FUNCTION_BLOCK Unifilar_HMI (* Service Interface Function Block Type *)
  (* Standard: 61499-2 *)
  (* Version 0.0, 21/04/2026, template *)
  PACKAGE Hidryco.HidrycoLib;
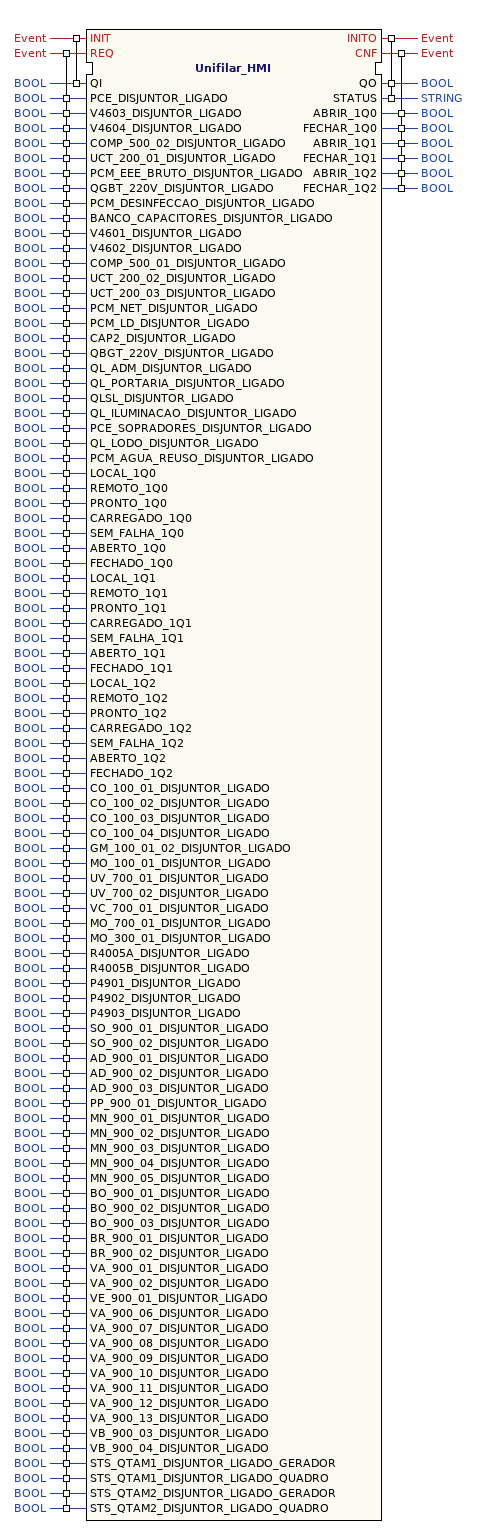
  EVENT_INPUT
    INIT WITH QI;
    REQ WITH PCE_DISJUNTOR_LIGADO, V4603_DISJUNTOR_LIGADO, V4604_DISJUNTOR_LIGADO, COMP_500_02_DISJUNTOR_LIGADO, UCT_200_01_DISJUNTOR_LIGADO, PCM_EEE_BRUTO_DISJUNTOR_LIGADO, QGBT_220V_DISJUNTOR_LIGADO, PCM_DESINFECCAO_DISJUNTOR_LIGADO, BANCO_CAPACITORES_DISJUNTOR_LIGADO, V4601_DISJUNTOR_LIGADO, V4602_DISJUNTOR_LIGADO, COMP_500_01_DISJUNTOR_LIGADO, UCT_200_02_DISJUNTOR_LIGADO, UCT_200_03_DISJUNTOR_LIGADO, PCM_NET_DISJUNTOR_LIGADO, PCM_LD_DISJUNTOR_LIGADO, CAP2_DISJUNTOR_LIGADO, QBGT_220V_DISJUNTOR_LIGADO, QL_ADM_DISJUNTOR_LIGADO, QL_PORTARIA_DISJUNTOR_LIGADO, QLSL_DISJUNTOR_LIGADO, QL_ILUMINACAO_DISJUNTOR_LIGADO, PCE_SOPRADORES_DISJUNTOR_LIGADO, QL_LODO_DISJUNTOR_LIGADO, PCM_AGUA_REUSO_DISJUNTOR_LIGADO, LOCAL_1Q0, REMOTO_1Q0, PRONTO_1Q0, CARREGADO_1Q0, SEM_FALHA_1Q0, ABERTO_1Q0, FECHADO_1Q0, LOCAL_1Q1, REMOTO_1Q1, PRONTO_1Q1, CARREGADO_1Q1, SEM_FALHA_1Q1, ABERTO_1Q1, FECHADO_1Q1, LOCAL_1Q2, REMOTO_1Q2, PRONTO_1Q2, CARREGADO_1Q2, SEM_FALHA_1Q2, ABERTO_1Q2, FECHADO_1Q2, CO_100_01_DISJUNTOR_LIGADO, CO_100_02_DISJUNTOR_LIGADO, CO_100_03_DISJUNTOR_LIGADO, CO_100_04_DISJUNTOR_LIGADO, GM_100_01_02_DISJUNTOR_LIGADO, MO_100_01_DISJUNTOR_LIGADO, UV_700_01_DISJUNTOR_LIGADO, UV_700_02_DISJUNTOR_LIGADO, VC_700_01_DISJUNTOR_LIGADO, MO_700_01_DISJUNTOR_LIGADO, MO_300_01_DISJUNTOR_LIGADO, R4005A_DISJUNTOR_LIGADO, R4005B_DISJUNTOR_LIGADO, P4901_DISJUNTOR_LIGADO, P4902_DISJUNTOR_LIGADO, P4903_DISJUNTOR_LIGADO, SO_900_01_DISJUNTOR_LIGADO, SO_900_02_DISJUNTOR_LIGADO, AD_900_01_DISJUNTOR_LIGADO, AD_900_02_DISJUNTOR_LIGADO, AD_900_03_DISJUNTOR_LIGADO, PP_900_01_DISJUNTOR_LIGADO, MN_900_01_DISJUNTOR_LIGADO, MN_900_02_DISJUNTOR_LIGADO, MN_900_03_DISJUNTOR_LIGADO, MN_900_04_DISJUNTOR_LIGADO, MN_900_05_DISJUNTOR_LIGADO, BO_900_01_DISJUNTOR_LIGADO, BO_900_02_DISJUNTOR_LIGADO, BO_900_03_DISJUNTOR_LIGADO, BR_900_01_DISJUNTOR_LIGADO, BR_900_02_DISJUNTOR_LIGADO, VA_900_01_DISJUNTOR_LIGADO, VA_900_02_DISJUNTOR_LIGADO, VE_900_01_DISJUNTOR_LIGADO, VA_900_06_DISJUNTOR_LIGADO, VA_900_07_DISJUNTOR_LIGADO, VA_900_08_DISJUNTOR_LIGADO, VA_900_09_DISJUNTOR_LIGADO, VA_900_10_DISJUNTOR_LIGADO, VA_900_11_DISJUNTOR_LIGADO, VA_900_12_DISJUNTOR_LIGADO, VA_900_13_DISJUNTOR_LIGADO, VB_900_03_DISJUNTOR_LIGADO, VB_900_04_DISJUNTOR_LIGADO, STS_QTAM1_DISJUNTOR_LIGADO_GERADOR, STS_QTAM1_DISJUNTOR_LIGADO_QUADRO, STS_QTAM2_DISJUNTOR_LIGADO_GERADOR, STS_QTAM2_DISJUNTOR_LIGADO_QUADRO;
  END_EVENT
  EVENT_OUTPUT
    INITO WITH QO, STATUS;
    CNF WITH ABRIR_1Q0, FECHAR_1Q0, ABRIR_1Q1, FECHAR_1Q1, ABRIR_1Q2, FECHAR_1Q2;
  END_EVENT
  VAR_INPUT
    QI : BOOL;
    PCE_DISJUNTOR_LIGADO : BOOL;
    V4603_DISJUNTOR_LIGADO : BOOL;
    V4604_DISJUNTOR_LIGADO : BOOL;
    COMP_500_02_DISJUNTOR_LIGADO : BOOL;
    UCT_200_01_DISJUNTOR_LIGADO : BOOL;
    PCM_EEE_BRUTO_DISJUNTOR_LIGADO : BOOL;
    QGBT_220V_DISJUNTOR_LIGADO : BOOL;
    PCM_DESINFECCAO_DISJUNTOR_LIGADO : BOOL;
    BANCO_CAPACITORES_DISJUNTOR_LIGADO : BOOL;
    V4601_DISJUNTOR_LIGADO : BOOL;
    V4602_DISJUNTOR_LIGADO : BOOL;
    COMP_500_01_DISJUNTOR_LIGADO : BOOL;
    UCT_200_02_DISJUNTOR_LIGADO : BOOL;
    UCT_200_03_DISJUNTOR_LIGADO : BOOL;
    PCM_NET_DISJUNTOR_LIGADO : BOOL;
    PCM_LD_DISJUNTOR_LIGADO : BOOL;
    CAP2_DISJUNTOR_LIGADO : BOOL;
    QBGT_220V_DISJUNTOR_LIGADO : BOOL;
    QL_ADM_DISJUNTOR_LIGADO : BOOL;
    QL_PORTARIA_DISJUNTOR_LIGADO : BOOL;
    QLSL_DISJUNTOR_LIGADO : BOOL;
    QL_ILUMINACAO_DISJUNTOR_LIGADO : BOOL;
    PCE_SOPRADORES_DISJUNTOR_LIGADO : BOOL;
    QL_LODO_DISJUNTOR_LIGADO : BOOL;
    PCM_AGUA_REUSO_DISJUNTOR_LIGADO : BOOL;
    LOCAL_1Q0 : BOOL;
    REMOTO_1Q0 : BOOL;
    PRONTO_1Q0 : BOOL;
    CARREGADO_1Q0 : BOOL;
    SEM_FALHA_1Q0 : BOOL;
    ABERTO_1Q0 : BOOL;
    FECHADO_1Q0 : BOOL;
    LOCAL_1Q1 : BOOL;
    REMOTO_1Q1 : BOOL;
    PRONTO_1Q1 : BOOL;
    CARREGADO_1Q1 : BOOL;
    SEM_FALHA_1Q1 : BOOL;
    ABERTO_1Q1 : BOOL;
    FECHADO_1Q1 : BOOL;
    LOCAL_1Q2 : BOOL;
    REMOTO_1Q2 : BOOL;
    PRONTO_1Q2 : BOOL;
    CARREGADO_1Q2 : BOOL;
    SEM_FALHA_1Q2 : BOOL;
    ABERTO_1Q2 : BOOL;
    FECHADO_1Q2 : BOOL;
    CO_100_01_DISJUNTOR_LIGADO : BOOL;
    CO_100_02_DISJUNTOR_LIGADO : BOOL;
    CO_100_03_DISJUNTOR_LIGADO : BOOL;
    CO_100_04_DISJUNTOR_LIGADO : BOOL;
    GM_100_01_02_DISJUNTOR_LIGADO : BOOL;
    MO_100_01_DISJUNTOR_LIGADO : BOOL;
    UV_700_01_DISJUNTOR_LIGADO : BOOL;
    UV_700_02_DISJUNTOR_LIGADO : BOOL;
    VC_700_01_DISJUNTOR_LIGADO : BOOL;
    MO_700_01_DISJUNTOR_LIGADO : BOOL;
    MO_300_01_DISJUNTOR_LIGADO : BOOL;
    R4005A_DISJUNTOR_LIGADO : BOOL;
    R4005B_DISJUNTOR_LIGADO : BOOL;
    P4901_DISJUNTOR_LIGADO : BOOL;
    P4902_DISJUNTOR_LIGADO : BOOL;
    P4903_DISJUNTOR_LIGADO : BOOL;
    SO_900_01_DISJUNTOR_LIGADO : BOOL;
    SO_900_02_DISJUNTOR_LIGADO : BOOL;
    AD_900_01_DISJUNTOR_LIGADO : BOOL;
    AD_900_02_DISJUNTOR_LIGADO : BOOL;
    AD_900_03_DISJUNTOR_LIGADO : BOOL;
    PP_900_01_DISJUNTOR_LIGADO : BOOL;
    MN_900_01_DISJUNTOR_LIGADO : BOOL;
    MN_900_02_DISJUNTOR_LIGADO : BOOL;
    MN_900_03_DISJUNTOR_LIGADO : BOOL;
    MN_900_04_DISJUNTOR_LIGADO : BOOL;
    MN_900_05_DISJUNTOR_LIGADO : BOOL;
    BO_900_01_DISJUNTOR_LIGADO : BOOL;
    BO_900_02_DISJUNTOR_LIGADO : BOOL;
    BO_900_03_DISJUNTOR_LIGADO : BOOL;
    BR_900_01_DISJUNTOR_LIGADO : BOOL;
    BR_900_02_DISJUNTOR_LIGADO : BOOL;
    VA_900_01_DISJUNTOR_LIGADO : BOOL;
    VA_900_02_DISJUNTOR_LIGADO : BOOL;
    VE_900_01_DISJUNTOR_LIGADO : BOOL;
    VA_900_06_DISJUNTOR_LIGADO : BOOL;
    VA_900_07_DISJUNTOR_LIGADO : BOOL;
    VA_900_08_DISJUNTOR_LIGADO : BOOL;
    VA_900_09_DISJUNTOR_LIGADO : BOOL;
    VA_900_10_DISJUNTOR_LIGADO : BOOL;
    VA_900_11_DISJUNTOR_LIGADO : BOOL;
    VA_900_12_DISJUNTOR_LIGADO : BOOL;
    VA_900_13_DISJUNTOR_LIGADO : BOOL;
    VB_900_03_DISJUNTOR_LIGADO : BOOL;
    VB_900_04_DISJUNTOR_LIGADO : BOOL;
    STS_QTAM1_DISJUNTOR_LIGADO_GERADOR : BOOL;
    STS_QTAM1_DISJUNTOR_LIGADO_QUADRO : BOOL;
    STS_QTAM2_DISJUNTOR_LIGADO_GERADOR : BOOL;
    STS_QTAM2_DISJUNTOR_LIGADO_QUADRO : BOOL;
  END_VAR
  VAR_OUTPUT
    QO : BOOL; (* Event Output Qualifier *)
    STATUS : STRING; (* Service Status *)
    ABRIR_1Q0 : BOOL;
    FECHAR_1Q0 : BOOL;
    ABRIR_1Q1 : BOOL;
    FECHAR_1Q1 : BOOL;
    ABRIR_1Q2 : BOOL;
    FECHAR_1Q2 : BOOL;
  END_VAR
  SERVICE /
    SEQUENCE 
    END_SEQUENCE
  END_SERVICE
END_FUNCTION_BLOCK
